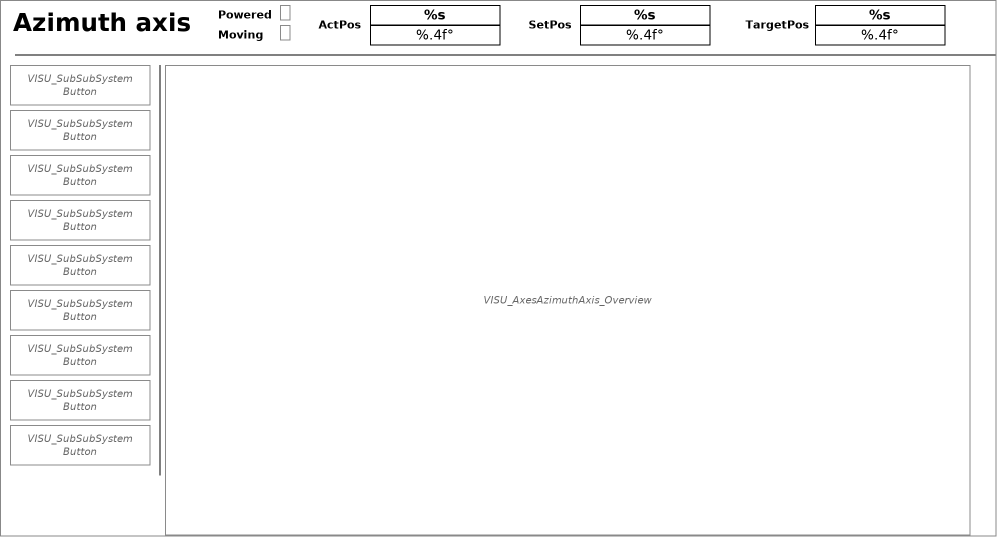
VISUALIZATION VISU_AxesAzimuthAxis  // 997x537
VAR_IN_OUT
	ref : AxesAzimuthAxis;
    ref_aziDriveChannel : AX52XXDriveChannel;
    ref_ablDriveChannel : AX52XXDriveChannel;
    widget : AxesAzimuthAxisWidget;
END_VAR
    Rectangle (10,0 195x45), "Azimuth axis"
    Frame (10,65 140x40)
        shows VISU_SubSubSystemButton(widget := widget.button_overview)
        OnMouseClick: FrameSelectionChange Selection=SelectedFrame=26eb0533-0645-4710-820d-78aa3cb40b18, GlobSel=AssignType=Directly, SelType=Locally
        OnMouseClick: execute { widget.activeTab := AxesAzimuthAxisTabs.OVERVIEW; }
    Frame (165,65 805x470)
        shows VISU_AxesAzimuthAxis_Overview(ref := ref, widget := widget)
        shows VISU_AxesAzimuthAxis_Processes(ref := ref, ref_aziDriveChannel := ref_aziDriveChannel, widget := widget)
        shows VISU_AX522DriveChannel(ref := ref_aziDriveChannel, widget := widget.aziDriveChannel)
        shows VISU_AX522DriveChannel(ref := ref_ablDriveChannel, widget := widget.ablDriveChannel)
        shows VISU_AngularAxis(axis := ref.parts.virtualAxis, widget := widget.virtualAxis)
        shows VISU_AngularAxis(axis := ref.parts.physicalAxis, widget := widget.physicalAxis)
        shows VISU_AngularAxis(axis := ref.parts.ablAxis, widget := widget.ablAxis)
        shows VISU_AxesAzimuthAxis_Lidas(ref := ref, widget := widget)
        shows VISU_AxesAzimuthAxis_AbsoluteEncoder(ref := ref, widget := widget)
        p4174417010: ref.parts.virtualAxis
        p2620823199: ref
    Line (160,475) (160,65)
    Frame (10,155 140x40)
        shows VISU_SubSubSystemButton(widget := widget.button_aziDriveChannel)
        OnMouseClick: FrameSelectionChange Selection=SelectedFrame=26eb0533-0645-4710-820d-78aa3cb40b18, Selection=2, GlobSel=AssignType=Directly, SelType=Locally
        OnMouseClick: execute { widget.activeTab := AxesAzimuthAxisTabs.AZI_DRIVE_CHANNEL; }
    Frame (10,200 140x40)
        shows VISU_SubSubSystemButton(widget := widget.button_ablDriveChannel)
        OnMouseClick: FrameSelectionChange Selection=SelectedFrame=26eb0533-0645-4710-820d-78aa3cb40b18, Selection=3, GlobSel=AssignType=Directly, SelType=Locally
        OnMouseClick: execute { widget.activeTab := AxesAzimuthAxisTabs.ABL_DRIVE_CHANNEL; }
    Frame (10,245 140x40)
        shows VISU_SubSubSystemButton(widget := widget.button_virtualAxis)
        OnMouseClick: FrameSelectionChange Selection=SelectedFrame=26eb0533-0645-4710-820d-78aa3cb40b18, Selection=4, GlobSel=AssignType=Directly, SelType=Locally
        OnMouseClick: execute { widget.activeTab := AxesAzimuthAxisTabs.VIRTUAL_AXIS; }
    Frame (10,290 140x40)
        shows VISU_SubSubSystemButton(widget := widget.button_physicalAxis)
        OnMouseClick: FrameSelectionChange Selection=SelectedFrame=26eb0533-0645-4710-820d-78aa3cb40b18, Selection=5, GlobSel=AssignType=Directly, SelType=Locally
        OnMouseClick: execute { widget.activeTab := AxesAzimuthAxisTabs.PHYSICAL_AXIS; }
    Frame (10,335 140x40)
        shows VISU_SubSubSystemButton(widget := widget.button_ablAxis)
        OnMouseClick: FrameSelectionChange Selection=SelectedFrame=26eb0533-0645-4710-820d-78aa3cb40b18, Selection=6, GlobSel=AssignType=Directly, SelType=Locally
        OnMouseClick: execute { widget.activeTab := AxesAzimuthAxisTabs.ABL_AXIS; }
    Frame (10,380 140x40)
        shows VISU_SubSubSystemButton(widget := widget.button_lidas)
        OnMouseClick: FrameSelectionChange Selection=SelectedFrame=26eb0533-0645-4710-820d-78aa3cb40b18, Selection=7, GlobSel=AssignType=Directly, SelType=Locally
        OnMouseClick: execute { widget.activeTab := AxesAzimuthAxisTabs.LIDAS; }
    Frame (10,425 140x40)
        shows VISU_SubSubSystemButton(widget := widget.button_absoluteEncoder)
        OnMouseClick: FrameSelectionChange Selection=SelectedFrame=26eb0533-0645-4710-820d-78aa3cb40b18, Selection=8, GlobSel=AssignType=Directly, SelType=Locally
        OnMouseClick: execute { widget.activeTab := AxesAzimuthAxisTabs.ABSOLUTE_ENCODER; }
    Frame (10,110 140x40)
        shows VISU_SubSubSystemButton(widget := widget.button_processes)
        OnMouseClick: FrameSelectionChange Selection=SelectedFrame=26eb0533-0645-4710-820d-78aa3cb40b18, Selection=1, GlobSel=AssignType=Directly, SelType=Locally
        OnMouseClick: execute { widget.activeTab := AxesAzimuthAxisTabs.PROCESSES; }
    Line (995,55) (15,55)
    Label (310,0 60x50), "ActPos"
    Rectangle (370,5 130x20), "%s", text variable: widget.actPos.dmsString
    Rectangle (370,25 130x20), "%.4f°", text variable: ref.actPos.degrees.value
    Label (520,0 60x50), "SetPos"
    Rectangle (580,5 130x20), "%s", text variable: widget.setPos.dmsString
    Rectangle (580,25 130x20), "%.4f°", text variable: ref.setPos.degrees.value
    Label (740,0 75x50), "TargetPos"
    Rectangle (815,5 130x20), "%s", text variable: widget.targetPos.dmsString
    Rectangle (815,25 130x20), "%.4f°", text variable: ref.targetPos.degrees.value
    Label (215,5 65x20), "Powered"
    Frame (280,5 10x15)
        shows VISU_State_gray_green(state := ref.statuses.poweredStatus.enabled)
    Label (215,25 65x20), "Moving"
    Frame (280,25 10x15)
        shows VISU_State_gray_green(state := ref.parts.physicalAxis.axis_ref.Status.Moving)
END_VISUALIZATION

(* stored: Version 1.1.0.1, ProductVersion 3.1.4019.2
   Visu VISU_AxesAzimuthAxis: Id {cefbc39a-fa90-48b0-9fab-e6bc52162ef2} *)
